// Mitsubishi GX Works2 project: 2022래더도   PLC: Q03UDV

PROGRAM MAIN
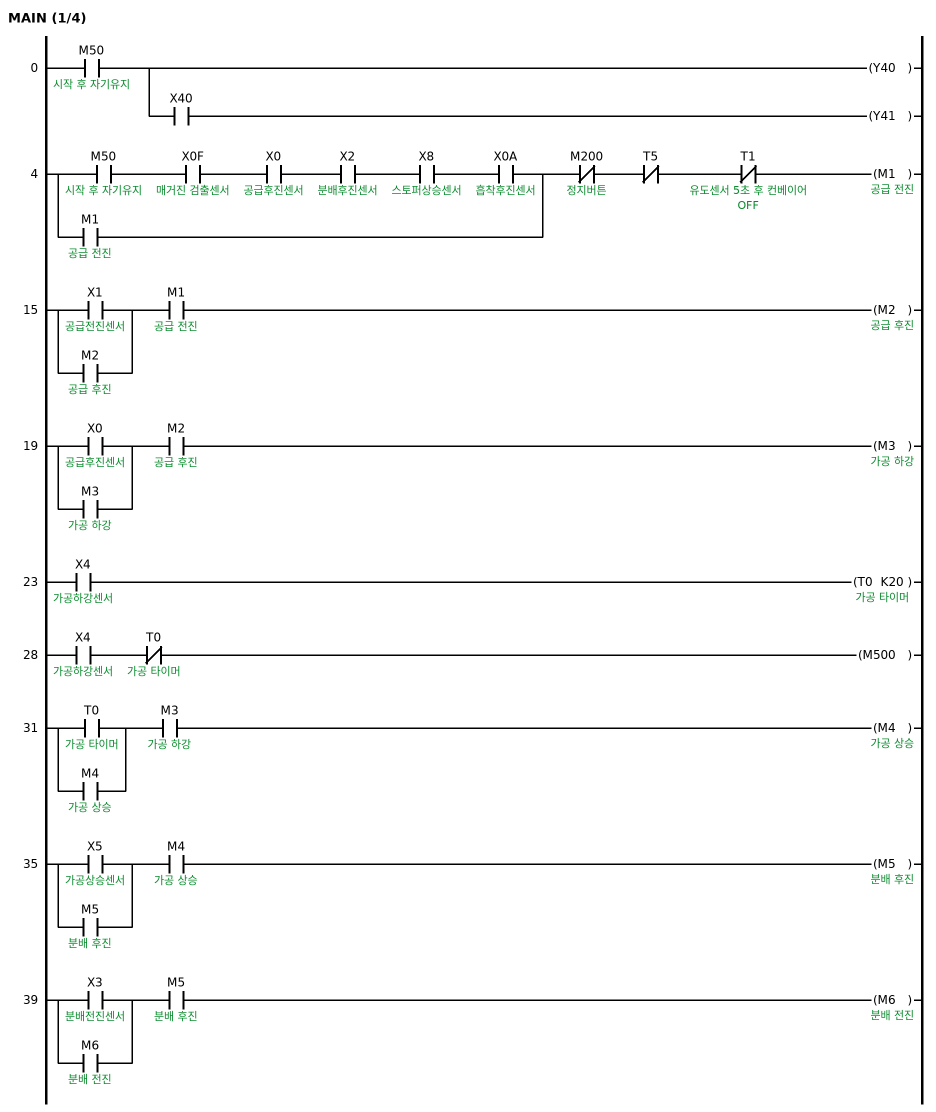
0     LD      M50  ; 시작 후 자기유지
      OUT     Y40
      AND     X40
      OUT     Y41
4     LD      M50  ; 시작 후 자기유지
      AND     X0F  ; 매거진 검출센서
      AND     X0  ; 공급후진센서
      AND     X2  ; 분배후진센서
      AND     X8  ; 스토퍼상승센서
      AND     X0A  ; 흡착후진센서
      OR      M1  ; 공급 전진
      ANI     M200  ; 정지버튼
      ANI     T5
      ANI     T1  ; 유도센서 5초 후 컨베이어 OFF
      OUT     M1  ; 공급 전진
15    LD      X1  ; 공급전진센서
      OR      M2  ; 공급 후진
      AND     M1  ; 공급 전진
      OUT     M2  ; 공급 후진
19    LD      X0  ; 공급후진센서
      OR      M3  ; 가공 하강
      AND     M2  ; 공급 후진
      OUT     M3  ; 가공 하강
23    LD      X4  ; 가공하강센서
      OUT     T0 K20  ; 가공 타이머
28    LD      X4  ; 가공하강센서
      ANI     T0  ; 가공 타이머
      OUT     M500
31    LD      T0  ; 가공 타이머
      OR      M4  ; 가공 상승
      AND     M3  ; 가공 하강
      OUT     M4  ; 가공 상승
35    LD      X5  ; 가공상승센서
      OR      M5  ; 분배 후진
      AND     M4  ; 가공 상승
      OUT     M5  ; 분배 후진
39    LD      X3  ; 분배전진센서
      OR      M6  ; 분배 전진
      AND     M5  ; 분배 후진
      OUT     M6  ; 분배 전진
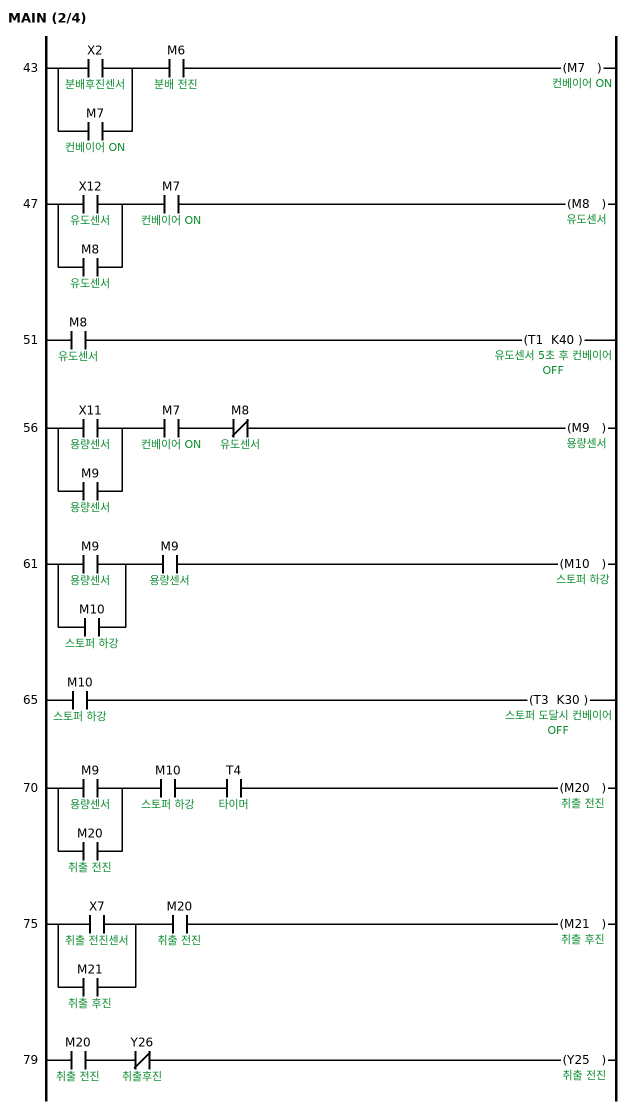
43    LD      X2  ; 분배후진센서
      OR      M7  ; 컨베이어 ON
      AND     M6  ; 분배 전진
      OUT     M7  ; 컨베이어 ON
47    LD      X12  ; 유도센서
      OR      M8  ; 유도센서
      AND     M7  ; 컨베이어 ON
      OUT     M8  ; 유도센서
51    LD      M8  ; 유도센서
      OUT     T1 K40  ; 유도센서 5초 후 컨베이어 OFF
56    LD      X11  ; 용량센서
      OR      M9  ; 용량센서
      AND     M7  ; 컨베이어 ON
      ANI     M8  ; 유도센서
      OUT     M9  ; 용량센서
61    LD      M9  ; 용량센서
      OR      M10  ; 스토퍼 하강
      AND     M9  ; 용량센서
      OUT     M10  ; 스토퍼 하강
65    LD      M10  ; 스토퍼 하강
      OUT     T3 K30  ; 스토퍼 도달시 컨베이어 OFF
70    LD      M9  ; 용량센서
      OR      M20  ; 취출 전진
      AND     M10  ; 스토퍼 하강
      AND     T4  ; 타이머
      OUT     M20  ; 취출 전진
75    LD      X7  ; 취출 전진센서
      OR      M21  ; 취출 후진
      AND     M20  ; 취출 전진
      OUT     M21  ; 취출 후진
79    LD      M20  ; 취출 전진
      ANI     Y26  ; 취출후진
      OUT     Y25  ; 취출 전진
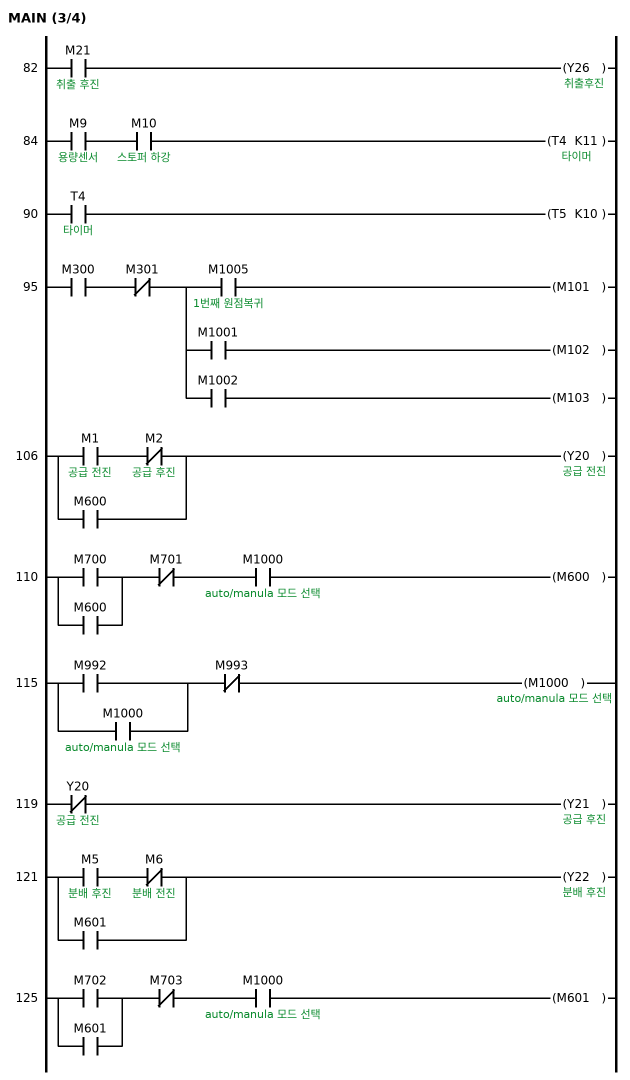
82    LD      M21  ; 취출 후진
      OUT     Y26  ; 취출후진
84    LD      M9  ; 용량센서
      AND     M10  ; 스토퍼 하강
      OUT     T4 K11  ; 타이머
90    LD      T4  ; 타이머
      OUT     T5 K10
95    LD      M300
      ANI     M301
      MPS
      AND     M1005  ; 1번째 원점복귀
      OUT     M101
      MRD
      AND     M1001
      OUT     M102
      MPP
      AND     M1002
      OUT     M103
106   LD      M1  ; 공급 전진
      ANI     M2  ; 공급 후진
      OR      M600
      OUT     Y20  ; 공급 전진
110   LD      M700
      OR      M600
      ANI     M701
      AND     M1000  ; auto/manula 모드 선택
      OUT     M600
115   LD      M992
      OR      M1000  ; auto/manula 모드 선택
      ANI     M993
      OUT     M1000  ; auto/manula 모드 선택
119   LDI     Y20  ; 공급 전진
      OUT     Y21  ; 공급 후진
121   LD      M5  ; 분배 후진
      ANI     M6  ; 분배 전진
      OR      M601
      OUT     Y22  ; 분배 후진
125   LD      M702
      OR      M601
      ANI     M703
      AND     M1000  ; auto/manula 모드 선택
      OUT     M601
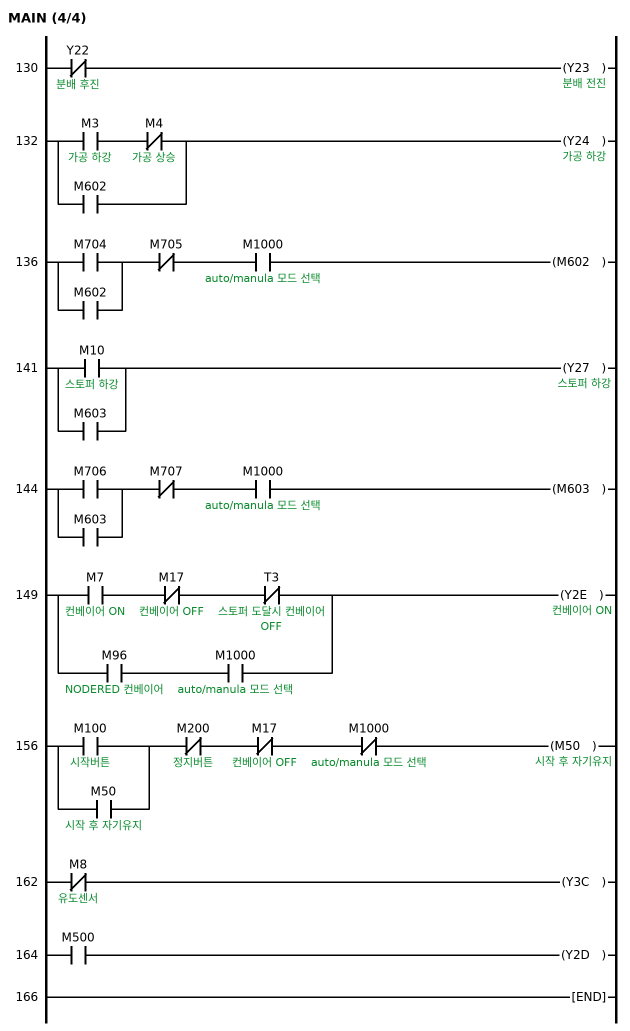
130   LDI     Y22  ; 분배 후진
      OUT     Y23  ; 분배 전진
132   LD      M3  ; 가공 하강
      ANI     M4  ; 가공 상승
      OR      M602
      OUT     Y24  ; 가공 하강
136   LD      M704
      OR      M602
      ANI     M705
      AND     M1000  ; auto/manula 모드 선택
      OUT     M602
141   LD      M10  ; 스토퍼 하강
      OR      M603
      OUT     Y27  ; 스토퍼 하강
144   LD      M706
      OR      M603
      ANI     M707
      AND     M1000  ; auto/manula 모드 선택
      OUT     M603
149   LD      M7  ; 컨베이어 ON
      ANI     M17  ; 컨베이어 OFF
      ANI     T3  ; 스토퍼 도달시 컨베이어 OFF
      LD      M96  ; NODERED 컨베이어
      AND     M1000  ; auto/manula 모드 선택
      ORB
      OUT     Y2E  ; 컨베이어 ON
156   LD      M100  ; 시작버튼
      OR      M50  ; 시작 후 자기유지
      ANI     M200  ; 정지버튼
      ANI     M17  ; 컨베이어 OFF
      ANI     M1000  ; auto/manula 모드 선택
      OUT     M50  ; 시작 후 자기유지
162   LDI     M8  ; 유도센서
      OUT     Y3C
164   LD      M500
      OUT     Y2D
166   END
END_PROGRAM

// device comments not shown above
X9  ; 스토퍼 하강센서
X13  ; 스토퍼검출센서
X18  ; UR3 동작완료
X1E  ; 정지버튼 (PB2)
X1F  ; 시작버튼 (PB1)
Y30  ; uram 동작완료
Y31  ; ur3 화이트
Y32  ; ur3 블랙
Y33  ; ur3 레드
M11  ; 영상계측 시작
M12  ; 영상계측결과-화이트
M14  ; 로봇팔동작-화이트
M15  ; 로봇팔동작-블랙
M16  ; 로봇팔 동작 완료
M18  ; 로봇팔 동작 -레드
M19  ; UR3시작신호
M31  ; UR3 화이트동작
M32  ; UR3 블랙동작
M33  ; UR3 레드 동작
T2  ; 스토퍼 하강 후 딜레이
T7  ; 스토퍼 타이머
